// TIA Portal V17 export
// export: Created 2025-06-26T06:49:22.6581315Z, ExportSetting WithDefaults, DisplayName Totally Integrated Automation Portal, DisplayVersion V17 Update 8, DisplayName TIA Portal Openness, DisplayVersion V17 Update 8, DisplayName TIA Portal Version Control Interface, DisplayVersion V17, DisplayName STEP 7 Professional, DisplayVersion V17 Update 8, DisplayName STEP 7 Safety, DisplayVersion V17 Update 6, DisplayName WinCC Advanced, DisplayVersion V17 Update 8
DATA_BLOCK "DB_Valves"   // DB46
{ S7_Optimized_Access := 'FALSE' }
AUTHOR : Heaten
VERSION : 0.1
// stored: AutoNumber false, DBAccessibleFromOPCUA true, IsOnlyStoredInLoadMemory false, IsWriteProtectedInAS false
   VAR RETAIN
      GH117_815 { S7_SetPoint := 'True'} : "stRegulatingValve";   // Dampfventil Kondensator ein
      GH117_821 { S7_SetPoint := 'True'} : "stRegulatingValve";   // Kondensatventil Kondensator aus
      GH117_812 { S7_SetPoint := 'True'} : "stRegulatingValve";   // Kondensatventil Verdampfer ein
      GH117_818 { S7_SetPoint := 'True'} : "stRegulatingValve";   // Dampfventil Verdampfer aus
   END_VAR
BEGIN
   GH117_815.Cmd.Position.Raw.iMin := 0;
   GH117_815.Cmd.Position.Raw.iMax := 1000;
   GH117_815.Cmd.Position.Eng.fMin := 0.0;
   GH117_815.Cmd.Position.Eng.fMax := 100.0;
   GH117_821.Cmd.Position.Raw.iMin := 0;
   GH117_821.Cmd.Position.Raw.iMax := 1000;
   GH117_821.Cmd.Position.Eng.fMin := 0.0;
   GH117_821.Cmd.Position.Eng.fMax := 100.0;
   GH117_812.Cmd.Position.Raw.iMin := 0;
   GH117_812.Cmd.Position.Raw.iMax := 1000;
   GH117_812.Cmd.Position.Eng.fMin := 0.0;
   GH117_812.Cmd.Position.Eng.fMax := 100.0;
   GH117_818.Cmd.Position.Raw.iMin := 0;
   GH117_818.Cmd.Position.Raw.iMax := 1000;
   GH117_818.Cmd.Position.Eng.fMin := 0.0;
   GH117_818.Cmd.Position.Eng.fMax := 100.0;
END_DATA_BLOCK
